// TIA Portal V20 export
ORGANIZATION_BLOCK "Main"   // OB1, FBD, ProgramCycle
TITLE = "Main Program Sweep (Cycle)"
{ S7_Optimized_Access := 'TRUE' }
// stored: SetENOAutomatically false
   VAR_INPUT
      Initial_Call : Bool;   // Initial call of this OB
      Remanence : Bool;   // =True, if remanent data are available
   END_VAR
   VAR_TEMP
      EV_CLASS : Byte;   // Bits 0-3 = 1:Coming event, Bits 4-7 = 1:Event class 1
      SCAN_1 : Byte;   // 1:Initial call of the OB, 3: Call 2-n of the OB
      PRIORITY : Byte;   // Priority of OB Execution
      OB_NUMBR : Byte;   // OB number
      RESERVED_1 : Byte;   // Reserved for system
      RESERVED_2 : Byte;   // Reserved for system
      PREV_CYCLE : Int;   // Previous program cycle time (milliseconds)
      MIN_CYCLE : Int;   // Minimum program cycle time (milliseconds)
      MAX_CYCLE : Int;   // Maximum program cycle time (milliseconds)
      DATE_TIME : Date_And_Time;   // Date and time OB started
      tempLreal : LReal;
   END_VAR
   VAR_TEMP   // added for the SCL form of the ladder/FBD networks
      _w1 : Bool;
      _s5time1 : S5Time;
      _w2 : Bool;
      _s5time2 : S5Time;
   END_VAR
BEGIN

NETWORK
TITLE = restart
      A     "firstScan";
      L     s5t#2s;
      SD    "T0";
      A     "T0";
      R     "firstScan";

NETWORK
TITLE = true/false test1/test0
      AN    "true";
      S     "true";
      A     "false";
      R     "false";

      AN    "test1";
      S     "test1";
      A     "test0";
      R     "test0";

      AN    "test1ibn";
      S     "test1ibn";
      A     "test0ibn";
      R     "test0ibn";


NETWORK
TITLE = clocks
      L     "systemClockByte";
      T     "clockByte";

      L     "cycleFlag";
      L     1;
      +I;
      T     "cycleFlag";

REGION Network 4: if you will test safety areas let run the plant in slow speed an set this tag
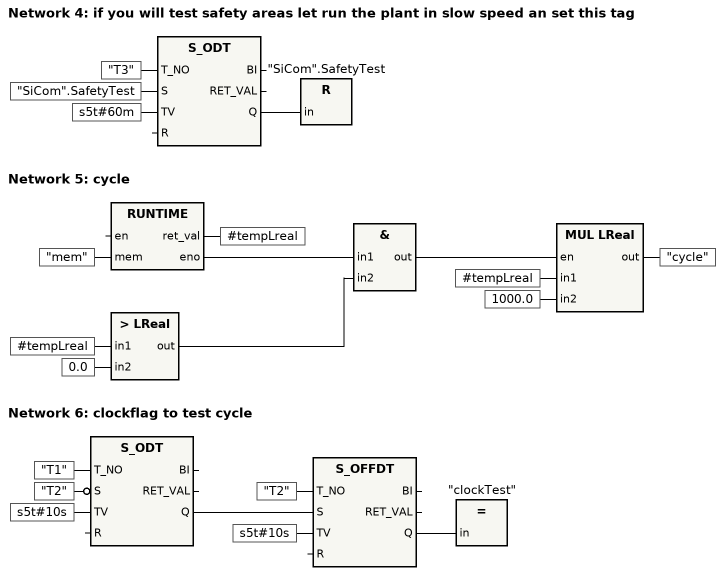
   #_s5time1 := S_ODT(T_NO := "T3", S := "SiCom".SafetyTest, TV := s5t#60m, Q => #_w1);
   IF #_w1 THEN "SiCom".SafetyTest := FALSE; END_IF;
END_REGION

REGION Network 5: cycle
   // no SCL statement known for Runtime: written as a call
   // ENO of a box is taken as its EN; it also drops when the box reports an error
   #tempLreal := Runtime(mem := "mem");
   IF #tempLreal > 0.0 THEN "cycle" := #tempLreal * 1000.0; END_IF;
END_REGION

REGION Network 6: clockflag to test cycle
   #_s5time1 := S_ODT(T_NO := "T1", S := NOT "T2", TV := s5t#10s, Q => #_w1);
   #_s5time2 := S_OFFDT(T_NO := "T2", S := #_w1, TV := s5t#10s, Q => #_w2);
   "clockTest" := #_w2;
END_REGION

NETWORK
TITLE = call instance

// Safety
      CALL  "SafetyCom", "SafetyCom_DB";

// Communication
      CALL  "Com", "Com_DB";

// General
      CALL  "Clock", "Clock_DB";
      CALL  "AutoIndication", "AutoIndication_DB";
      CALL  "Fault", "Fault_DB";
      CALL  "TestIo", "TestIo_DB";
      CALL  "ErrCom", "ErrCom_DB";

// Goldeneye
      CALL  "DataTakeOver", "DataTakeOver_DB";
      CALL  "Sensors", "Sensors_DB";
      CALL  "AdjScanner", "AdjScanner_DB";
      CALL  "AdjTop", "AdjTop_DB";
      CALL  "AdjLeft", "AdjLeft_DB";
      CALL  "AdjRight", "AdjRight_DB";
      CALL  "BlowOffValve", "BlowOffValve_DB";
      CALL  "AirConditioner", "AirConditioner_DB";

END_ORGANIZATION_BLOCK
